// Converts a size value to a position value.
FUNCTION F_SizeToPosition : T_Position // The position value corresponding to the given size.
VAR_INPUT
	Size : T_Size; // The size value to be converted to a position value.
END_VAR

F_SizeToPosition := Size;

END_FUNCTION

(* stored: Version 1.1.0.1
   POU F_SizeToPosition: Id {f3bae6ff-1672-07b4-0659-f8cd33d8bd24}, SpecialFunc None *)
